KUKA KRL program: Calibration_8.src

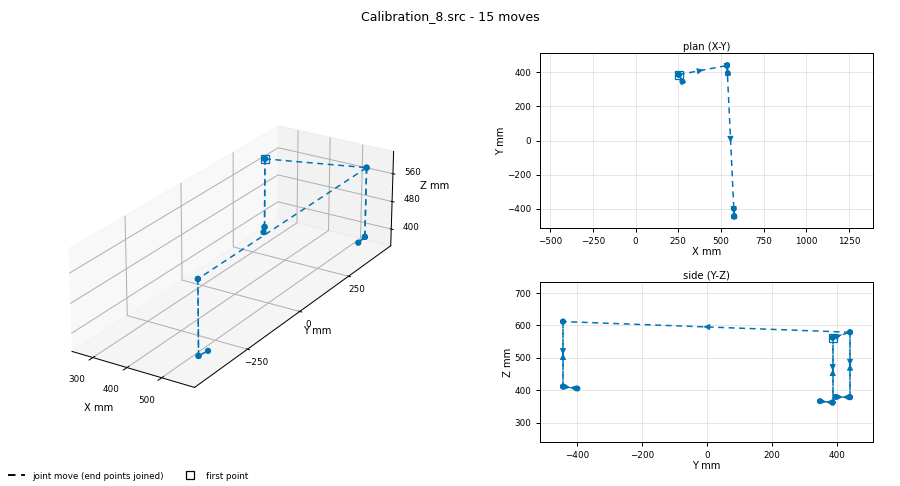
[picture p0: tool path of Calibration_8.src, 15 of 17 moves have a stored position in this frame; points joined in program order, loops and branches not executed]
&ACCESS RVP
&REL 1
&PARAM TEMPLATE = C:\KRC\Roboter\Template\vorgabe
&PARAM EDITMASK = *
DEF Calibration_8 ( )


;FOLD INI
;FOLD BASISTECH INI
GLOBAL INTERRUPT DECL 3 WHEN $STOPMESS==TRUE DO IR_STOPM ( )
INTERRUPT ON 3
BAS (#INITMOV,0 )
;ENDFOLD (BASISTECH INI)
;ENDFOLD (INI)

;FOLD STARTPOSITION - BASE IS 0, TOOL IS 5, SPEED IS 15%, POSITION IS A1 5,A2 -90,A3 100,A4 5,A5 -10,A6 -5,E1 0,E2 0,E3 0,E4 0
$BWDSTART = FALSE
PDAT_ACT = {VEL 15,ACC 100,APO_DIST 50}
FDAT_ACT = {TOOL_NO 5,BASE_NO 0,IPO_FRAME #BASE}
BAS (#PTP_PARAMS,15)
PTP  {A1 5,A2 -90,A3 100,A4 5,A5 -10,A6 -5,E1 0,E2 0,E3 0,E4 0}
;ENDFOLD

;FOLD LIN SPEED IS 0.1 m/sec, INTERPOLATION SETTINGS IN FOLD
$VEL.CP=0.1
$ADVANCE=3
;ENDFOLD

BAS(#VEL_PTP,10)
PTP {X 253.149, Y 386.192, Z 562.754, A -62.303, B -5.433, C -87.868, E1 0, E2 0, E3 0, E4 0, S 'B010'} C_PTP
PTP {X 253.149, Y 386.192, Z 362.754, A -62.303, B -5.433, C -87.868, E1 0, E2 0, E3 0, E4 0, S 'B010'} C_PTP
BAS(#VEL_PTP,2)
PTP {X 273.971, Y 346.527, Z 367.015, A -62.303, B -5.433, C -87.868, E1 0, E2 0, E3 0, E4 0, S 'B010'}
BAS(#VEL_PTP,10)
PTP {X 253.149, Y 386.192, Z 362.754, A -62.303, B -5.433, C -87.868, E1 0, E2 0, E3 0, E4 0, S 'B010'} C_PTP
PTP {X 253.149, Y 386.192, Z 562.754, A -62.303, B -5.433, C -87.868, E1 0, E2 0, E3 0, E4 0, S 'B010'} C_PTP
PTP {X 535.674, Y 439.555, Z 579.174, A -83.827, B -1.051, C -99.568, E1 0, E2 0, E3 0, E4 0, S 'B010'} C_PTP
PTP {X 535.674, Y 439.555, Z 379.174, A -83.827, B -1.051, C -99.568, E1 0, E2 0, E3 0, E4 0, S 'B010'} C_PTP
BAS(#VEL_PTP,2)
PTP {X 540.512, Y 394.823, Z 380, A -83.827, B -1.051, C -99.568, E1 0, E2 0, E3 0, E4 0, S 'B010'}
BAS(#VEL_PTP,10)
PTP {X 535.674, Y 439.555, Z 379.174, A -83.827, B -1.051, C -99.568, E1 0, E2 0, E3 0, E4 0, S 'B010'} C_PTP
PTP {X 535.674, Y 439.555, Z 579.174, A -83.827, B -1.051, C -99.568, E1 0, E2 0, E3 0, E4 0, S 'B010'} C_PTP
PTP {X 577.705, Y -444.332, Z 612.012, A 92.789, B 7.792, C 179.232, E1 0, E2 0, E3 0, E4 0, S 'B010'} C_PTP
PTP {X 577.705, Y -444.332, Z 412.012, A 92.789, B 7.792, C 179.232, E1 0, E2 0, E3 0, E4 0, S 'B010'} C_PTP
BAS(#VEL_PTP,2)
PTP {X 575.536, Y -399.8, Z 405.911, A 92.789, B 7.792, C 179.232, E1 0, E2 0, E3 0, E4 0, S 'B010'}
BAS(#VEL_PTP,10)
PTP {X 577.705, Y -444.332, Z 412.012, A 92.789, B 7.792, C 179.232, E1 0, E2 0, E3 0, E4 0, S 'B010'} C_PTP
PTP {X 577.705, Y -444.332, Z 612.012, A 92.789, B 7.792, C 179.232, E1 0, E2 0, E3 0, E4 0, S 'B010'} C_PTP
PTP {A1 5, A2 -90, A3 100, A4 5, A5 -10, A6 -5, E1 0, E2 0, E3 0, E4 0} C_PTP

END
